Fanuc KAREL source: kx00022.KL

-- PROVISIONAL review KL for V1013-1; original PC SHA256 45f1035b561ffdfdbb5bde5e230f4d3a0dfd39c9e22e9aad42cc854323f12e2c
-- Incomplete behavior may be omitted. Consult companion uncertainty JSON. Do not deploy.
PROGRAM KX00022
%NOLOCKGROUP
VAR
  I : INTEGER
  J : INTEGER
  B : BOOLEAN
  F : FILE
  S : STRING[80]
-- UNRESOLVED_DECL P type=000102
-- UNRESOLVED_DECL BA type=002012
BEGIN
  -- UNRESOLVED_PC offsets 5-15; opcodes 9D,22,9D,33,35
  -- UNRESOLVED_PC offsets 20-35; opcodes 22,9D,33,34,23
  -- UNRESOLVED_PC offsets 40-44; opcodes 7F
END KX00022
